TEXTLIST TL_Direction
  0 = 'Choose'
  1 = 'Input Module'
  2 = 'Output Module'
   = ''
END_TEXTLIST

(* stored: Version 1.1.0.1, ProductVersion 3.1.4020.3
   TextList TL_Direction: Id {705072db-12b3-437a-b8e9-cb8910e5414a} *)
